TYPE ST_HmiCommands :
STRUCT
    bStart                 : BOOL;
    bStop                  : BOOL;
    bReset                 : BOOL;
    bAcknowledge           : BOOL;
    bManualRequest         : BOOL;
    bIndexerManualEnable   : BOOL;
    bManualIndexForward    : BOOL;
    bManualIndexHome       : BOOL;
    bManualMainDoorUnlock  : BOOL;
	ePowerCmd              : E_PLC_Power := E_PLC_Power.Idle;

    // Main-screen operator/nest light toggle.
    // Physical output: Term 9 EL2809 Ch6 (bNestLight).
    bOperatorLight          : BOOL := TRUE;

    stHeatStakeTemperatureSettings : ST_HeatStakeTemperatureSettings;
    bApplyHeatStakeTemperatureSettings : BOOL;
    stHeatStakeProcessSettings : ST_HeatStakeProcessSettings;
	
	// =====================================================
	// Patch Dispensing Manual Mode
	// =====================================================
	
	bPatchManualEnable              : BOOL;
	
	bPatchSupportExtendRequest      : BOOL;
	bPatchSupportRetractRequest     : BOOL;
	
	bPatchVerticalUpRequest         : BOOL;
	bPatchVerticalDownRequest       : BOOL;
	
	bPatchDispenseRequest           : BOOL;
	bPatchAirBlowRequest            : BOOL;
	
	bPatchManualHomeRequest         : BOOL;
	bPatchManualRunSequence         : BOOL;

	// =====================================================
    // Heat Stake Manual Mode
	// =====================================================
	
    bHeatStakeManualEnable        : BOOL;
    bHeatStakeManualStakePatch    : BOOL;
    bHeatStakeManualUnlock        : BOOL;
    bHeatStakeManualLock          : BOOL;
    bHeatStakeManualHeadDown      : BOOL;
    bHeatStakeManualHeadUp        : BOOL;
    bHeatStakeManualSupportUp     : BOOL;

	// =====================================================
	// Vision Manual Mode
	// =====================================================
	
	bVisionManualEnable                	: BOOL;
	
	bVisionHorizontalBackRequest       	: BOOL;
	bVisionHorizontalFrontRequest      	: BOOL;
	
	bVisionVerticalUpRequest           	: BOOL;
	bVisionVerticalIntermediateRequest 	: BOOL;
	bVisionVerticalFullDownRequest     	: BOOL;
	
	bVisionGripOpenRequest             	: BOOL;
	bVisionGripCloseRequest            	: BOOL;
	
	bVisionRotate0Request              	: BOOL;
	bVisionRotate180Request            	: BOOL;
	
	bVisionSupportExtendRequest        	: BOOL;
	bVisionManualRunSequence 			: BOOL;
	
	bVisionManualHomeRequest 			: BOOL;

	
    // Nest settings command buffer. Every change is persisted automatically.
    aNestEnabled : ARRAY[1..4] OF BOOL := [TRUE, TRUE, TRUE, TRUE];

    // Popup OK acknowledgement.
    bAcknowledgeDisabledNestPartPopup 	: BOOL;
	bReprocessPopupAcknowledge 			: BOOL;
    bAcknowledgeRejectChuteFull 		: BOOL;

    uiResetStatisticsNestId				: UINT;
	
	
END_STRUCT
END_TYPE

(* stored: Version 1.1.0.1, ProductVersion 3.1.4026.18
   DUT ST_HmiCommands: Id {cea0711c-b7bf-4958-9705-69290143acac} *)
